// TIA Portal V19 export
DATA_BLOCK "OB82_DB"   // DB82
{ S7_Optimized_Access := 'TRUE' }
// stored: AutoNumber false, MemoryReserve 0
   VAR RETAIN
      vars : "OB82_vars";
      ComponentDiag : DIS;
      SubComponentDiag : DNN;
   END_VAR
BEGIN
END_DATA_BLOCK
